// TIA Portal V20 export
FUNCTION "GetTransaction_ID" : Void   // FC20222, LAD
{ S7_Optimized_Access := 'TRUE' }
// stored: AutoNumber false, SetENOAutomatically false
   VAR_INPUT
      i_Start : Int;
   END_VAR
   VAR_OUTPUT
      oTransactionID : DWord;
   END_VAR
   VAR_TEMP
      i_Dummy : Int;
      t_DTL : DTL;
      tDTL_String : String;
      tDTL_LInt : LInt;
   END_VAR
   VAR_TEMP   // added for the SCL form of the ladder/FBD networks
      _w1 : Bool;
      _w2 : Bool;
      _w3 : Bool;
      _w4 : Bool;
      _w5 : Bool;
      _w6 : Bool;
   END_VAR
BEGIN

REGION Network 1: Read time of day
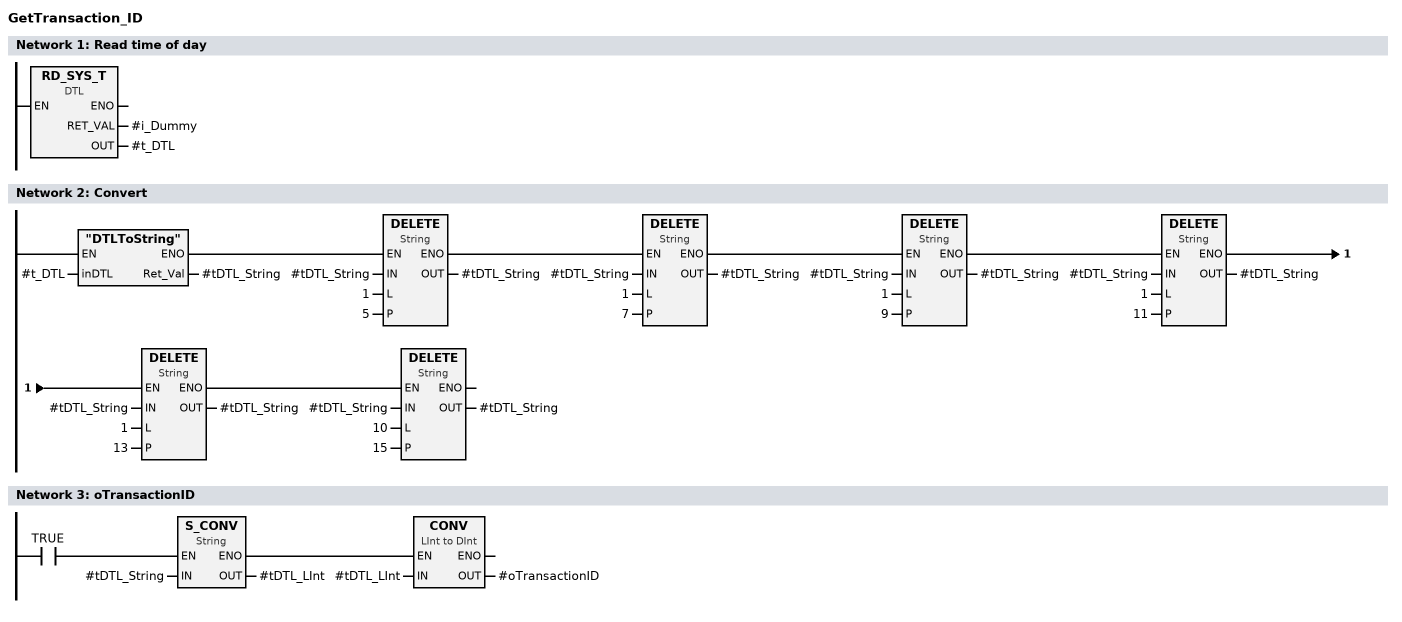
   RUNG wire#powerrail
      { S7_Templates := "date_type := DTL" } RD_SYS_T(RET_VAL => #i_Dummy, OUT => #t_DTL)
   END_RUNG
   // the same network as SCL:
   #i_Dummy := RD_SYS_T(OUT => #t_DTL);
END_REGION

REGION Network 2: Convert
   RUNG wire#powerrail
      "DTLToString"(inDTL := #t_DTL, Ret_Val => #tDTL_String)
      { S7_Templates := "str_type := String" } DELETE(IN := #tDTL_String, L := 1, P := 5, OUT => #tDTL_String)
      { S7_Templates := "str_type := String" } DELETE(IN := #tDTL_String, L := 1, P := 7, OUT => #tDTL_String)
      { S7_Templates := "str_type := String" } DELETE(IN := #tDTL_String, L := 1, P := 9, OUT => #tDTL_String)
      { S7_Templates := "str_type := String" } DELETE(IN := #tDTL_String, L := 1, P := 11, OUT => #tDTL_String)
      { S7_Templates := "str_type := String" } DELETE(IN := #tDTL_String, L := 1, P := 13, OUT => #tDTL_String)
      { S7_Templates := "str_type := String" } DELETE(IN := #tDTL_String, L := 10, P := 15, OUT => #tDTL_String)
   END_RUNG
   // the same network as SCL:
   #tDTL_String := "DTLToString"(inDTL := #t_DTL, ENO => #_w1);
   DELETE(EN := #_w1, IN := #tDTL_String, L := 1, P := 5, OUT => #tDTL_String, ENO => #_w2);
   DELETE(EN := #_w2, IN := #tDTL_String, L := 1, P := 7, OUT => #tDTL_String, ENO => #_w3);
   DELETE(EN := #_w3, IN := #tDTL_String, L := 1, P := 9, OUT => #tDTL_String, ENO => #_w4);
   DELETE(EN := #_w4, IN := #tDTL_String, L := 1, P := 11, OUT => #tDTL_String, ENO => #_w5);
   DELETE(EN := #_w5, IN := #tDTL_String, L := 1, P := 13, OUT => #tDTL_String, ENO => #_w6);
   IF #_w6 THEN DELETE(IN := #tDTL_String, L := 10, P := 15, OUT => #tDTL_String); END_IF;
END_REGION

REGION Network 3: oTransactionID
   RUNG wire#powerrail
      Contact( TRUE )
      { S7_Templates := "[src_type := String, dest_type := LInt]" } S_CONV(IN := #tDTL_String, OUT => #tDTL_LInt)
      { S7_Templates := "[SrcType := LInt, DestType := DInt]" } Convert(in := #tDTL_LInt, out => #oTransactionID)
   END_RUNG
   // the same network as SCL:
   S_CONV(EN := TRUE, IN := #tDTL_String, OUT => #tDTL_LInt, ENO => #_w1);
   IF #_w1 THEN #oTransactionID := LINT_TO_DINT(#tDTL_LInt); END_IF;
END_REGION
END_FUNCTION
